FUNCTION_BLOCK EventLogger
VAR
	EventBuffer : ARRAY[1..EVENT_BUFFER_MAX_SIZE] OF ST_Event;
	CurrentEventBufferIndex : INT := 0;
	_PersistentEventStorage : I_PersistentEventStorage;
END_VAR
VAR CONSTANT
	EVENT_BUFFER_MAX_SIZE : INT := 100;
END_VAR

METHOD PUBLIC AddEvent : BOOL
VAR_INPUT
	eEventType : E_EventType;
	eEventSeverity : TcEventSeverity;
	nEventIdentity : UDINT;
	sEventText : STRING(255);
END_VAR
IF NOT IsEventBufferFull() THEN
	//todo
	CurrentEventBufferIndex := CurrentEventBufferIndex + 1;
	EventBuffer[CurrentEventBufferIndex].eEventType := eEventType;
	EventBuffer[CurrentEventBufferIndex].eEventSeverity := eEventSeverity;
	EventBuffer[CurrentEventBufferIndex].nEventIdentity := nEventIdentity;
	EventBuffer[CurrentEventBufferIndex].sEventText := sEventText;
	F_UpdateEventTimestampWithSystemTime(stEvent := EventBuffer[CurrentEventBufferIndex]); 
	AddEvent := TRUE;
ELSE
	AddEvent := FALSE;
END_IF

_PersistentEventStorage.StoreEvent(stEvent := EventBuffer[CurrentEventBufferIndex]);
END_METHOD

METHOD FB_Init : BOOL
VAR_INPUT
	bInitRetains : BOOL;
	bInCopyCode : BOOL;
	iPersistentEventStorage : I_PersistentEventStorage;
END_VAR
_PersistentEventStorage := iPersistentEventStorage;
END_METHOD

METHOD PRIVATE IsEventBufferFull : BOOL
IF (CurrentEventBufferIndex + 1) >= EVENT_BUFFER_MAX_SIZE THEN
	IsEventBufferFull := TRUE;
ELSE
	IsEventBufferFull := FALSE;
END_IF
END_METHOD

END_FUNCTION_BLOCK

(* stored: Version 1.1.0.1, ProductVersion 3.1.4024.12
   POU EventLogger: Id {49a270de-7b38-4c0a-b542-93db06ca3178}, SpecialFunc None
   Method AddEvent: Id {8442e16c-f730-4c65-b703-9df028836144}
   Method FB_Init: Id {732d1647-b707-4d0e-b915-0e3d09f67b76}
   Method IsEventBufferFull: Id {6c0e3054-2059-437d-ace7-75813699a690} *)
